// TwinCAT 3 PLC project Adaptor_Pattern
// ProgramVersion: 3.1.4024.0
// libraries:
//   Tc2_Standard, * (Beckhoff Automation GmbH)
//   Tc2_System, * (Beckhoff Automation GmbH)
//   Tc3_Module, * (Beckhoff Automation GmbH)
// project tree:
//   3rd Party Library/Interfaces/ ITF_MQTTTool.TcIO
//   3rd Party Library/ mqttCommunication.TcPOU
//   Adaptor/ mqttCommsAdaptor.TcPOU
//   Classes/ ADSDataService.TcPOU, ITF_MachineDataService.TcIO, MachineControl.TcPOU
//   / PlcTask.TcTTO
//   POUs/ MAIN.TcPOU
// (motion and I/O tree: see PLC project simple_factory_pattern)
// real-time tasks:
//   TASK PlcTask: cycle T#10ms, priority 20, ADS port 350
//   TASK PlcTask1: cycle T#10ms, priority 21, ADS port 351
//   TASK PlcTask2: cycle T#10ms, priority 22, ADS port 352
//   TASK PlcTask3: cycle T#10ms, priority 23, ADS port 353
//   TASK PlcTask4: cycle T#10ms, priority 24, ADS port 354
//   TASK PlcTask5: cycle T#10ms, priority 25, ADS port 355
//   TASK PlcTask6: cycle T#10ms, priority 26, ADS port 356
//   TASK PlcTask7: cycle T#10ms, priority 27, ADS port 357

CONFIGURATION Adaptor_Pattern
    RESOURCE PLC ON TwinCAT3
        TASK PlcTask(INTERVAL := T#10ms, PRIORITY := 27);
        PROGRAM MAIN WITH PlcTask : MAIN;
    END_RESOURCE
END_CONFIGURATION

// ---- 3rd Party Library/Interfaces/ITF_MQTTTool.TcIO
INTERFACE ITF_MQTTTool

METHOD SendMQTTMessage : BOOL
VAR_INPUT
	Status : STRING;
END_VAR
END_METHOD

END_INTERFACE

// ---- Classes/ITF_MachineDataService.TcIO
INTERFACE ITF_MachineDataService

METHOD SendStatus : INT
VAR_INPUT
	Status : INT;
END_VAR
END_METHOD

END_INTERFACE

// ---- POUs/MAIN.TcPOU
PROGRAM MAIN
VAR
	dataService : ADSDataService;
	newDataService : mqttCommsAdaptor;
	myMachine : MachineControl := (DataService := newDataService);
	sendStatusRequest: BOOL;
END_VAR

IF sendStatusRequest THEN
	sendStatusRequest := FALSE;
	myMachine.PushMachineStatus();
END_IF

END_PROGRAM

// ---- Classes/ADSDataService.TcPOU
FUNCTION_BLOCK ADSDataService IMPLEMENTS ITF_MachineDataService
VAR
	_messageSent : int;
END_VAR

METHOD SendStatus : INT
VAR_INPUT
	Status : INT;
END_VAR
_messageSent := Status;
END_METHOD

END_FUNCTION_BLOCK

// ---- Adaptor/mqttCommsAdaptor.TcPOU
FUNCTION_BLOCK mqttCommsAdaptor IMPLEMENTS ITF_MachineDataService
VAR
	mqttComms : mqttCommunication;
END_VAR

METHOD SendStatus : INT
VAR_INPUT
	Status	: INT;
END_VAR
mqttComms.SendMQTTMessage(Status := TO_STRING(Status));
END_METHOD

END_FUNCTION_BLOCK

// ---- 3rd Party Library/mqttCommunication.TcPOU
FUNCTION_BLOCK mqttCommunication IMPLEMENTS ITF_MQTTTool
VAR
	_messageSent : string;
END_VAR

METHOD SendMQTTMessage : BOOL
VAR_INPUT
	Status : STRING;
END_VAR
_messageSent := Status;
END_METHOD

END_FUNCTION_BLOCK

// ---- Classes/MachineControl.TcPOU
FUNCTION_BLOCK MachineControl
VAR
	_dataService : ITF_MachineDataService;
	MyStatus : INT := 3;
END_VAR

PROPERTY DataService : ITF_MachineDataService
GET
DataService := _dataService;
END_GET
SET
_dataService := DataService;
END_SET
END_PROPERTY

METHOD PushMachineStatus : INT
VAR_INPUT
END_VAR
_dataService.SendStatus(MyStatus);
END_METHOD

END_FUNCTION_BLOCK
